TYPE ST_RecipeTypeStation : // Phisical Station
STRUCT
	nIdx	: UINT;
	bEnable	: BOOL;
	nActiveTestCount	: UINT; // can be any type of Leak Test for any mod. This is the total num of test the station has.
	nActiveAteqDevice	: UINT;
	nActiveValveBank	: UINT;
END_STRUCT
END_TYPE

(* stored: Version 1.1.0.1
   DUT ST_RecipeTypeStation: Id {109aca7e-36c5-06e5-032c-1e12f3e8c0a9} *)
